(* IEC 61131-3 sources: inj-machine-docs/docs/IM_SYS_PRG/Code/实例管理, 1 file *)

(* ---- Instances.st ---- *)
(*
  Instances.st
  功能：
  1. 定义整机仍需要在全局范围复用的顶层功能块实例。
  2. 顶层调度统一收口到 `PRG_MainControl`，因此这里只保留主入口真正需要的实例。

  说明：
  1. `FB_MachineController` 内部已经自行管理手动、调模、自动和各执行模块子实例。
  2. 温控块 `FB_EK312` 已提升到顶层，由 `PRG_MainControl` 直接调用。
  3. 旧版 `gvl_fbAutoCycle`、`gvl_fbManualMode`、`gvl_fbMoldAdjustMode` 已移除，避免重复调用。
*)
VAR_GLOBAL
    (* HMI 参数同步实例。 *)
    gvl_fbHMIParaInterface: FB_HMIParaInterface;   // 顶层唯一 HMI 参数同步实例，由 `PRG_MainControl` 每拍先调用。

    (* 顶层温控实例。 *)
    gvl_fbEK312: FB_EK312;                         // 顶层唯一温控实例，由 `PRG_MainControl` 直接调用，并与 `FB_MachineController` 保持完全分离。

    (* 机器级统一主控实例。 *)
    gvl_fbMachineController: FB_MachineController; // 顶层唯一机器主控实例，负责模式路由、模块调度和状态汇总。
END_VAR
